(*	SINT_T, USINT_T, INT_T, UINT_T, DINT_T, UDINT_T, 
				LINT_T, ULINT_T, REALT_T, LREAL_T*)
CASE TypeOfValue OF
	//VAR_TYPES.SINT_T:
	IBaseLibrary.TypeClass.TYPE_SINT:
		GetValueStringFaktor := SINT_TO_STRING(VALUE.SINT_T);
	//VAR_TYPES.USINT_T:
	IBaseLibrary.TypeClass.TYPE_USINT:
		GetValueStringFaktor := USINT_TO_STRING(VALUE.USINT_T);		
	//VAR_TYPES.INT_T:
	IBaseLibrary.TypeClass.TYPE_INT:
		GetValueStringFaktor := INT_TO_STRING(VALUE.INT_T);
	//VAR_TYPES.UINT_T:
	IBaseLibrary.TypeClass.TYPE_UINT:
		GetValueStringFaktor := UINT_TO_STRING(VALUE.UINT_T);
	//VAR_TYPES.DINT_T:
	IBaseLibrary.TypeClass.TYPE_DINT:
		GetValueStringFaktor := DINT_TO_STRING(VALUE.DINT_T);
	//VAR_TYPES.UDINT_T:
	IBaseLibrary.TypeClass.TYPE_UDINT:
		GetValueStringFaktor := UDINT_TO_STRING(VALUE.UDINT_T);
	//VAR_TYPES.LINT_T:
	IBaseLibrary.TypeClass.TYPE_LINT:
		GetValueStringFaktor := LINT_TO_STRING(VALUE.LINT_T);
	//VAR_TYPES.ULINT_T:
	IBaseLibrary.TypeClass.TYPE_ULINT:
		GetValueStringFaktor := ULINT_TO_STRING(VALUE.ULINT_T);
	//VAR_TYPES.REAL_T:
	IBaseLibrary.TypeClass.TYPE_REAL:
		GetValueStringFaktor := OSCAT_BASIC.REAL_TO_STRF(VALUE.REAL_T * RealFaktor,DecimalPlace,'.');
	//VAR_TYPES.LREAL_T:
	IBaseLibrary.TypeClass.TYPE_LREAL:
		GetValueStringFaktor := BASIC_Extension.LREAL_TO_STRF(VALUE.LREAL_T * RealFaktor,DecimalPlace,'.');
	//VAR_TYPES.BYTE_T:
	IBaseLibrary.TypeClass.TYPE_BYTE:
		GetValueStringFaktor := BYTE_TO_STRING(VALUE.BYTE_T);
	//VAR_TYPES.WORD_T:
	IBaseLibrary.TypeClass.TYPE_WORD:
		GetValueStringFaktor := WORD_TO_STRING(VALUE.WORD_T);
	//VAR_TYPES.DWORD_T:
	IBaseLibrary.TypeClass.TYPE_DWORD:
		GetValueStringFaktor := DWORD_TO_STRING(VALUE.DWORD_T);
	//VAR_TYPES.LWORD_T:
	IBaseLibrary.TypeClass.TYPE_LWORD:
		GetValueStringFaktor := LWORD_TO_STRING(VALUE.LWORD_T);
	//VAR_TYPES.DT_T:
	IBaseLibrary.TypeClass.TYPE_DATEANDTIME:
		GetValueStringFaktor := DT_TO_STRING(VALUE.DT_T);
	//VAR_TYPES.TIME_T:
	IBaseLibrary.TypeClass.TYPE_TIME:
		GetValueStringFaktor := TIME_TO_STRING(VALUE.TIME_T);
	//VAR_TYPES.LTIME_T:
	IBaseLibrary.TypeClass.TYPE_LTIME:
		GetValueStringFaktor := LTIME_TO_STRING(VALUE.LTIME_T);
	//VAR_TYPES.TOD_T:
	IBaseLibrary.TypeClass.TYPE_TIMEOFDAY:
		GetValueStringFaktor := TOD_TO_STRING(VALUE.TOD_T);
	//VAR_TYPES.BOOL_T:
	IBaseLibrary.TypeClass.TYPE_BOOL:
		GetValueStringFaktor := BOOL_TO_STRING(VALUE.BOOL_T);
	//VAR_TYPES.DATE_T:
	IBaseLibrary.TypeClass.TYPE_DATE:
		GetValueStringFaktor := DATE_TO_STRING(VALUE.DATE_T);
END_CASE

END_FUNCTION

// Common/Functions/unionAdd
FUNCTION unionAdd : ALL_TYPES_UNION
VAR_INPUT
	a:ALL_TYPES_UNION;
	b:ALL_TYPES_UNION;
	TypeOfValue:IBaseLibrary.TypeClass;
END_VAR
VAR
END_VAR

(*	SINT_T, USINT_T, INT_T, UINT_T, DINT_T, UDINT_T, 
				LINT_T, ULINT_T, REALT_T, LREAL_T*)
CASE TypeOfValue OF
	IBaseLibrary.TypeClass.TYPE_SINT:
		unionAdd.SINT_T := a.SINT_T + b.SINT_T;
	IBaseLibrary.TypeClass.TYPE_USINT:
		unionAdd.USINT_T := a.USINT_T + b.USINT_T;
	IBaseLibrary.TypeClass.TYPE_INT:
		unionAdd.INT_T := a.INT_T + b.INT_T;
	IBaseLibrary.TypeClass.TYPE_UINT:
		unionAdd.UINT_T := a.UINT_T + b.UINT_T;
	IBaseLibrary.TypeClass.TYPE_DINT:
		unionAdd.DINT_T := a.UINT_T + b.UINT_T;
	IBaseLibrary.TypeClass.TYPE_UDINT:
		unionAdd.UDINT_T := a.UDINT_T + b.UDINT_T;
	IBaseLibrary.TypeClass.TYPE_LINT:
		unionAdd.LINT_T := a.LINT_T + b.LINT_T;
	IBaseLibrary.TypeClass.TYPE_ULINT:
		unionAdd.ULINT_T := a.ULINT_T + b.ULINT_T;
	IBaseLibrary.TypeClass.TYPE_REAL:
		unionAdd.REAL_T := a.REAL_T + b.REAL_T;
	IBaseLibrary.TypeClass.TYPE_LREAL:
		unionAdd.LREAL_T := a.LREAL_T + b.LREAL_T;
	IBaseLibrary.TypeClass.TYPE_BYTE:
		unionAdd.BYTE_T := a.BYTE_T + b.BYTE_T;
	IBaseLibrary.TypeClass.TYPE_WORD:
		unionAdd.WORD_T := a.WORD_T + b.WORD_T;
	IBaseLibrary.TypeClass.TYPE_DWORD:
		unionAdd.DWORD_T := a.DWORD_T + b.DWORD_T;
	IBaseLibrary.TypeClass.TYPE_LWORD:
		unionAdd.LWORD_T := a.LWORD_T + b.LWORD_T;
	IBaseLibrary.TypeClass.TYPE_DATEANDTIME:
	{warning "need to implement"}
		//unionAdd.DT_T := a.DT_T + b.DT_T;
	IBaseLibrary.TypeClass.TYPE_TIME:
		unionAdd.TIME_T := a.TIME_T + b.TIME_T;
	IBaseLibrary.TypeClass.TYPE_LTIME:
		unionAdd.LTIME_T := a.LTIME_T + b.LTIME_T;
	IBaseLibrary.TypeClass.TYPE_TIMEOFDAY:
	{warning "need to implement"}
		//unionAdd.TOD_T := a.TOD_T + b.TOD_T;
	IBaseLibrary.TypeClass.TYPE_BOOL:
		unionAdd.BOOL_T := a.BOOL_T AND b.BOOL_T;
	IBaseLibrary.TypeClass.TYPE_DATE:
	{warning "need to implement"}
		//unionAdd.DATE_T := a.DATE_T + b.DATE_T;
	
END_CASE

END_FUNCTION

// Common/Functions/unionSub
FUNCTION unionSub : ALL_TYPES_UNION
VAR_INPUT
	a:ALL_TYPES_UNION;
	b:ALL_TYPES_UNION;
	TypeOfValue:IBaseLibrary.TypeClass;
END_VAR
VAR
END_VAR

(*	SINT_T, USINT_T, INT_T, UINT_T, DINT_T, UDINT_T, 
				LINT_T, ULINT_T, REALT_T, LREAL_T*)
CASE TypeOfValue OF
	IBaseLibrary.TypeClass.TYPE_SINT:
		unionSub.SINT_T := a.SINT_T - b.SINT_T;
	IBaseLibrary.TypeClass.TYPE_USINT:
		unionSub.USINT_T := a.USINT_T - b.USINT_T;
	IBaseLibrary.TypeClass.TYPE_INT:
		unionSub.INT_T := a.INT_T - b.INT_T;
	IBaseLibrary.TypeClass.TYPE_UINT:
		unionSub.UINT_T := a.UINT_T - b.UINT_T;
	IBaseLibrary.TypeClass.TYPE_DINT:
		unionSub.DINT_T := a.UINT_T - b.UINT_T;
	IBaseLibrary.TypeClass.TYPE_UDINT:
		unionSub.UDINT_T := a.UDINT_T - b.UDINT_T;
	IBaseLibrary.TypeClass.TYPE_LINT:
		unionSub.LINT_T := a.LINT_T - b.LINT_T;
	IBaseLibrary.TypeClass.TYPE_ULINT:
		unionSub.ULINT_T := a.ULINT_T - b.ULINT_T;
	IBaseLibrary.TypeClass.TYPE_REAL:
		unionSub.REAL_T := a.REAL_T - b.REAL_T;
	IBaseLibrary.TypeClass.TYPE_LREAL:
		unionSub.LREAL_T := a.LREAL_T - b.LREAL_T;
	IBaseLibrary.TypeClass.TYPE_BYTE:
		unionSub.BYTE_T := a.BYTE_T - b.BYTE_T;
	IBaseLibrary.TypeClass.TYPE_WORD:
		unionSub.WORD_T := a.WORD_T - b.WORD_T;
	IBaseLibrary.TypeClass.TYPE_DWORD:
		unionSub.DWORD_T := a.DWORD_T - b.DWORD_T;
	IBaseLibrary.TypeClass.TYPE_LWORD:
		unionSub.LWORD_T := a.LWORD_T - b.LWORD_T;
	IBaseLibrary.TypeClass.TYPE_DATEANDTIME:
	{warning "need to implement"}
		//unionSub.DT_T := a.DT_T - b.DT_T;
	IBaseLibrary.TypeClass.TYPE_TIME:
		unionSub.TIME_T := a.TIME_T - b.TIME_T;
	IBaseLibrary.TypeClass.TYPE_LTIME:
		unionSub.LTIME_T := a.LTIME_T - b.LTIME_T;
	IBaseLibrary.TypeClass.TYPE_TIMEOFDAY:
	{warning "need to implement"}
		//unionSub.TOD_T := a.TOD_T - b.TOD_T;
	IBaseLibrary.TypeClass.TYPE_BOOL:
		unionSub.BOOL_T := a.BOOL_T AND b.BOOL_T;
	IBaseLibrary.TypeClass.TYPE_DATE:
	{warning "need to implement"}
		//unionSub.DATE_T := a.DATE_T - b.DATE_T;
	
END_CASE

END_FUNCTION

// Common/Functions/unionMul
FUNCTION unionMul : ALL_TYPES_UNION
VAR_INPUT
	a:ALL_TYPES_UNION;
	b:ALL_TYPES_UNION;
	TypeOfValue:IBaseLibrary.TypeClass;
END_VAR
VAR
END_VAR

(*	SINT_T, USINT_T, INT_T, UINT_T, DINT_T, UDINT_T, 
				LINT_T, ULINT_T, REALT_T, LREAL_T*)
CASE TypeOfValue OF
	IBaseLibrary.TypeClass.TYPE_SINT:
		unionMul.SINT_T := a.SINT_T * b.SINT_T;
	IBaseLibrary.TypeClass.TYPE_USINT:
		unionMul.USINT_T := a.USINT_T * b.USINT_T;
	IBaseLibrary.TypeClass.TYPE_INT:
		unionMul.INT_T := a.INT_T * b.INT_T;
	IBaseLibrary.TypeClass.TYPE_UINT:
		unionMul.UINT_T := a.UINT_T * b.UINT_T;
	IBaseLibrary.TypeClass.TYPE_DINT:
		unionMul.DINT_T := a.UINT_T * b.UINT_T;
	IBaseLibrary.TypeClass.TYPE_UDINT:
		unionMul.UDINT_T := a.UDINT_T * b.UDINT_T;
	IBaseLibrary.TypeClass.TYPE_LINT:
		unionMul.LINT_T := a.LINT_T * b.LINT_T;
	IBaseLibrary.TypeClass.TYPE_ULINT:
		unionMul.ULINT_T := a.ULINT_T * b.ULINT_T;
	IBaseLibrary.TypeClass.TYPE_REAL:
		unionMul.REAL_T := a.REAL_T * b.REAL_T;
	IBaseLibrary.TypeClass.TYPE_LREAL:
		unionMul.LREAL_T := a.LREAL_T * b.LREAL_T;
	IBaseLibrary.TypeClass.TYPE_BYTE:
		unionMul.BYTE_T := a.BYTE_T * b.BYTE_T;
	IBaseLibrary.TypeClass.TYPE_WORD:
		unionMul.WORD_T := a.WORD_T * b.WORD_T;
	IBaseLibrary.TypeClass.TYPE_DWORD:
		unionMul.DWORD_T := a.DWORD_T * b.DWORD_T;
	IBaseLibrary.TypeClass.TYPE_LWORD:
		unionMul.LWORD_T := a.LWORD_T * b.LWORD_T;
	IBaseLibrary.TypeClass.TYPE_DATEANDTIME:
	{warning "need to implement"}
		//unionMul.DT_T := a.DT_T * b.DT_T;
	IBaseLibrary.TypeClass.TYPE_TIME:
	//unionMul.TOD_T := a.TOD_T * b.TOD_T;
		//unionMul.TIME_T := a.TIME_T * b.TIME_T;
	IBaseLibrary.TypeClass.TYPE_LTIME:
	//unionMul.TOD_T := a.TOD_T * b.TOD_T;
		//unionMul.LTIME_T := a.LTIME_T * b.LTIME_T;
	IBaseLibrary.TypeClass.TYPE_TIMEOFDAY:
	{warning "need to implement"}
		//unionMul.TOD_T := a.TOD_T * b.TOD_T;
	IBaseLibrary.TypeClass.TYPE_BOOL:
		unionMul.BOOL_T := a.BOOL_T AND b.BOOL_T;
	IBaseLibrary.TypeClass.TYPE_DATE:
	{warning "need to implement"}
		//unionMul.DATE_T := a.DATE_T * b.DATE_T;
	
END_CASE

END_FUNCTION

// Common/Functions/unionDiv
FUNCTION unionDiv : ALL_TYPES_UNION
VAR_INPUT
	a:ALL_TYPES_UNION;
	b:ALL_TYPES_UNION;
	TypeOfValue:IBaseLibrary.TypeClass;
END_VAR
VAR
END_VAR

(*	SINT_T, USINT_T, INT_T, UINT_T, DINT_T, UDINT_T, 
				LINT_T, ULINT_T, REALT_T, LREAL_T*)
CASE TypeOfValue OF
	IBaseLibrary.TypeClass.TYPE_SINT:
		unionDiv.SINT_T := a.SINT_T / b.SINT_T;
	IBaseLibrary.TypeClass.TYPE_USINT:
		unionDiv.USINT_T := a.USINT_T / b.USINT_T;
	IBaseLibrary.TypeClass.TYPE_INT:
		unionDiv.INT_T := a.INT_T / b.INT_T;
	IBaseLibrary.TypeClass.TYPE_UINT:
		unionDiv.UINT_T := a.UINT_T / b.UINT_T;
	IBaseLibrary.TypeClass.TYPE_DINT:
		unionDiv.DINT_T := a.UINT_T / b.UINT_T;
	IBaseLibrary.TypeClass.TYPE_UDINT:
		unionDiv.UDINT_T := a.UDINT_T / b.UDINT_T;
	IBaseLibrary.TypeClass.TYPE_LINT:
		unionDiv.LINT_T := a.LINT_T / b.LINT_T;
	IBaseLibrary.TypeClass.TYPE_ULINT:
		unionDiv.ULINT_T := a.ULINT_T / b.ULINT_T;
	IBaseLibrary.TypeClass.TYPE_REAL:
		unionDiv.REAL_T := a.REAL_T / b.REAL_T;
	IBaseLibrary.TypeClass.TYPE_LREAL:
		unionDiv.LREAL_T := a.LREAL_T / b.LREAL_T;
	IBaseLibrary.TypeClass.TYPE_BYTE:
		unionDiv.BYTE_T := a.BYTE_T / b.BYTE_T;
	IBaseLibrary.TypeClass.TYPE_WORD:
		unionDiv.WORD_T := a.WORD_T / b.WORD_T;
	IBaseLibrary.TypeClass.TYPE_DWORD:
		unionDiv.DWORD_T := a.DWORD_T / b.DWORD_T;
	IBaseLibrary.TypeClass.TYPE_LWORD:
		unionDiv.LWORD_T := a.LWORD_T / b.LWORD_T;
	IBaseLibrary.TypeClass.TYPE_DATEANDTIME:
	{warning "need to implement"}
		//unionDiv.DT_T := a.DT_T / b.DT_T;
	IBaseLibrary.TypeClass.TYPE_TIME:
	//unionDiv.TOD_T := a.TOD_T / b.TOD_T;
		//unionDiv.TIME_T := a.TIME_T / b.TIME_T;
	IBaseLibrary.TypeClass.TYPE_LTIME:
	//unionDiv.TOD_T := a.TOD_T / b.TOD_T;
		//unionDiv.LTIME_T := a.LTIME_T / b.LTIME_T;
	IBaseLibrary.TypeClass.TYPE_TIMEOFDAY:
	{warning "need to implement"}
		//unionDiv.TOD_T := a.TOD_T / b.TOD_T;
	IBaseLibrary.TypeClass.TYPE_BOOL:
		unionDiv.BOOL_T := a.BOOL_T AND b.BOOL_T;
	IBaseLibrary.TypeClass.TYPE_DATE:
	{warning "need to implement"}
		//unionDiv.DATE_T := a.DATE_T / b.DATE_T;
	
END_CASE

END_FUNCTION

// Common/Function Blocks/UpDown
FUNCTION_BLOCK UpDown
VAR_INPUT
	Start:BOOL;
	VarType:IBaseLibrary.TypeClass;
	faktor:UINT;
	Imp: BOOL;
	limitUp:REAL;
	limitDown:REAL;
END_VAR
VAR_IN_OUT
	Who:ALL_TYPES_UNION;
	
END_VAR
VAR_OUTPUT
END_VAR
VAR
	dir: BOOL;
	triggerStart:R_TRIG;
	diffVal:ALL_TYPES_UNION;
END_VAR

triggerStart(CLK := Start);
IF triggerStart.Q THEN
	dir := NOT dir;
END_IF

IF Start AND Imp THEN
	diffVal := uint_to_Union(value:= faktor, TypeOfValue:= VarType);
	IF dir THEN
		who := unionAdd(a:= Who, b:= diffVal, TypeOfValue:= VarType);
	ELSE
		who := unionSub(a:= Who, b:= diffVal, TypeOfValue:= VarType);
	END_IF
END_IF

END_FUNCTION_BLOCK

// Common/Functions/uint_to_Union
FUNCTION uint_to_Union : ALL_TYPES_UNION
VAR_INPUT
	TypeOfValue:IBaseLibrary.TypeClass;
	value:UINT;	

END_VAR
VAR
END_VAR

(*	SINT_T, USINT_T, INT_T, UINT_T, DINT_T, UDINT_T, 
				LINT_T, ULINT_T, REALT_T, LREAL_T*)
CASE TypeOfValue OF
	IBaseLibrary.TypeClass.TYPE_SINT:
		uint_to_Union.SINT_T := TO_SINT(value);
	IBaseLibrary.TypeClass.TYPE_USINT:
		uint_to_Union.USINT_T := TO_USINT(value);		
	IBaseLibrary.TypeClass.TYPE_INT:
		uint_to_Union.INT_T := TO_INT(value);
	IBaseLibrary.TypeClass.TYPE_UINT:
		uint_to_Union.UINT_T := TO_UINT(value);
	IBaseLibrary.TypeClass.TYPE_DINT:
		uint_to_Union.DINT_T := TO_DINT(value);
	IBaseLibrary.TypeClass.TYPE_UDINT:
		uint_to_Union.UDINT_T := TO_UDINT(value);
	IBaseLibrary.TypeClass.TYPE_LINT:
		AtomicWriteLInt(pDest:= ADR(uint_to_Union.LINT_T), liValue:= TO_LINT(value));
	IBaseLibrary.TypeClass.TYPE_ULINT:
		AtomicWriteULInt(pDest:= ADR(uint_to_Union.ULINT_T), uliValue:= TO_ULINT(value));
	IBaseLibrary.TypeClass.TYPE_REAL:
		uint_to_Union.REAL_T := TO_REAL(value);
	IBaseLibrary.TypeClass.TYPE_LREAL:
		AtomicWriteLReal(pDest:= ADR(uint_to_Union.LREAL_T), lrValue:= TO_LREAL(value));
	IBaseLibrary.TypeClass.TYPE_BYTE:
		uint_to_Union.BYTE_T := TO_BYTE(value);
	IBaseLibrary.TypeClass.TYPE_WORD:
		uint_to_Union.WORD_T := TO_WORD(value);
	IBaseLibrary.TypeClass.TYPE_DWORD:
		uint_to_Union.DWORD_T := TO_DWORD(value);
	IBaseLibrary.TypeClass.TYPE_LWORD:
		AtomicWriteLWord(pDest:= ADR(uint_to_Union.LWORD_T), lwValue:= TO_LWORD(value));
	IBaseLibrary.TypeClass.TYPE_DATEANDTIME:
		uint_to_Union.DT_T := TO_DT(value);
	IBaseLibrary.TypeClass.TYPE_TIME:
		uint_to_Union.TIME_T := TO_TIME(value);
	IBaseLibrary.TypeClass.TYPE_LTIME:
		AtomicWriteLTime(pDest:= ADR(uint_to_Union.LTIME_T), ltValue:= TO_LTIME(value));
	IBaseLibrary.TypeClass.TYPE_TIMEOFDAY:
		uint_to_Union.TOD_T := TO_TOD(value);
	IBaseLibrary.TypeClass.TYPE_BOOL:
		uint_to_Union.BOOL_T := TO_BOOL(value);
	IBaseLibrary.TypeClass.TYPE_DATE:
		uint_to_Union.DATE_T := TO_DATE(value);
	
	
END_CASE

END_FUNCTION

// Common/Functions/unionLimit
FUNCTION unionLimit : ALL_TYPES_UNION
VAR_INPUT
	in:ALL_TYPES_UNION;
	lMin:ALL_TYPES_UNION;
	lMax:ALL_TYPES_UNION;
	TypeOfValue:IBaseLibrary.TypeClass;
END_VAR
VAR
END_VAR

(*	SINT_T, USINT_T, INT_T, UINT_T, DINT_T, UDINT_T, 
				LINT_T, ULINT_T, REALT_T, LREAL_T*)
CASE TypeOfValue OF
	IBaseLibrary.TypeClass.TYPE_SINT:
		unionLimit.SINT_T := LIMIT(lMin.SINT_T, IN.SINT_T, lMax.SINT_T);
	IBaseLibrary.TypeClass.TYPE_USINT:
		unionLimit.USINT_T := LIMIT(lMin.USINT_T, IN.USINT_T, lMax.USINT_T);
	IBaseLibrary.TypeClass.TYPE_INT:
		unionLimit.INT_T := LIMIT(lMin.INT_T, IN.INT_T, lMax.INT_T);
	IBaseLibrary.TypeClass.TYPE_UINT:
		unionLimit.UINT_T := LIMIT(lMin.UINT_T, IN.UINT_T, lMax.UINT_T);
	IBaseLibrary.TypeClass.TYPE_DINT:
		unionLimit.DINT_T := LIMIT(lMin.DINT_T, IN.DINT_T, lMax.DINT_T);
	IBaseLibrary.TypeClass.TYPE_UDINT:
		unionLimit.UDINT_T := LIMIT(lMin.UDINT_T, IN.UDINT_T, lMax.UDINT_T);
	IBaseLibrary.TypeClass.TYPE_LINT:
		unionLimit.LINT_T := LIMIT(lMin.LINT_T, IN.LINT_T, lMax.LINT_T);
	IBaseLibrary.TypeClass.TYPE_ULINT:
		unionLimit.ULINT_T := LIMIT(lMin.ULINT_T, IN.ULINT_T, lMax.ULINT_T);
	IBaseLibrary.TypeClass.TYPE_REAL:
		unionLimit.REAL_T := LIMIT(lMin.REAL_T, IN.REAL_T, lMax.REAL_T);
	IBaseLibrary.TypeClass.TYPE_LREAL:
		unionLimit.LREAL_T := LIMIT(lMin.LREAL_T, IN.LREAL_T, lMax.LREAL_T);
	IBaseLibrary.TypeClass.TYPE_BYTE:
		unionLimit.BYTE_T := LIMIT(lMin.BYTE_T, IN.BYTE_T, lMax.BYTE_T);
	IBaseLibrary.TypeClass.TYPE_WORD:
		unionLimit.WORD_T := LIMIT(lMin.WORD_T, IN.WORD_T, lMax.WORD_T);
	IBaseLibrary.TypeClass.TYPE_DWORD:
		unionLimit.DWORD_T := LIMIT(lMin.DWORD_T, IN.DWORD_T, lMax.DWORD_T);
	IBaseLibrary.TypeClass.TYPE_LWORD:
		unionLimit.LWORD_T := LIMIT(lMin.LWORD_T, IN.LWORD_T, lMax.LWORD_T);
	IBaseLibrary.TypeClass.TYPE_DATEANDTIME:
		unionLimit.DT_T := LIMIT(lMin.DT_T, IN.DT_T, lMax.DT_T);
	IBaseLibrary.TypeClass.TYPE_TIME:
		unionLimit.TIME_T := LIMIT(lMin.TIME_T, IN.TIME_T, lMax.TIME_T);
	IBaseLibrary.TypeClass.TYPE_LTIME:
		unionLimit.LTIME_T := LIMIT(lMin.LTIME_T, IN.LTIME_T, lMax.LTIME_T);
	IBaseLibrary.TypeClass.TYPE_TIMEOFDAY:
		unionLimit.TOD_T := LIMIT(lMin.TOD_T, IN.TOD_T, lMax.TOD_T);
	IBaseLibrary.TypeClass.TYPE_BOOL:
		unionLimit.BOOL_T := LIMIT(lMin.BOOL_T, IN.BOOL_T, lMax.BOOL_T);
	IBaseLibrary.TypeClass.TYPE_DATE:
		unionLimit.DATE_T := LIMIT(lMin.DATE_T, IN.DATE_T, lMax.DATE_T);
	
END_CASE

END_FUNCTION

// Common/Functions/ScaleAllTypesUnion
FUNCTION ScaleAllTypesUnion : ALL_TYPES_UNION
VAR_INPUT
	in:ALL_TYPES_UNION;
	TypeOfVar:IBaseLibrary.TypeClass;
	I_LO : LREAL;
	I_HI : LREAL;
	O_LO : LREAL;
	O_HI : LREAL;
END_VAR
VAR

END_VAR

(*	SINT_T, USINT_T, INT_T, UINT_T, DINT_T, UDINT_T, 
				LINT_T, ULINT_T, REALT_T, LREAL_T*)
CASE TypeOfVar OF
	IBaseLibrary.TypeClass.TYPE_SINT:
		ScaleAllTypesUnion.SINT_T := TO_SINT(OSCAT_BASIC.SCALE_D(
			X:= TO_DWORD(in.SINT_T), I_LO:= TO_DWORD(I_LO), I_HI:= TO_DWORD(I_HI), O_LO:= TO_REAL(O_LO), O_HI:= TO_REAL(O_HI)));
	IBaseLibrary.TypeClass.TYPE_USINT:
		ScaleAllTypesUnion.USINT_T := TO_USINT(OSCAT_BASIC.SCALE_D(
			X:= TO_DWORD(in.USINT_T), I_LO:= TO_DWORD(I_LO), I_HI:= TO_DWORD(I_HI), O_LO:= TO_REAL(O_LO), O_HI:= TO_REAL(O_HI)));
	IBaseLibrary.TypeClass.TYPE_INT:
		ScaleAllTypesUnion.INT_T := TO_INT(OSCAT_BASIC.SCALE_D(
			X:= TO_DWORD(in.INT_T), I_LO:= TO_DWORD(I_LO), I_HI:= TO_DWORD(I_HI), O_LO:= TO_REAL(O_LO), O_HI:= TO_REAL(O_HI)));
	IBaseLibrary.TypeClass.TYPE_UINT:
		ScaleAllTypesUnion.UINT_T := TO_UINT(OSCAT_BASIC.SCALE_D(
			X:= TO_DWORD(in.UINT_T), I_LO:= TO_DWORD(I_LO), I_HI:= TO_DWORD(I_HI), O_LO:= TO_REAL(O_LO), O_HI:= TO_REAL(O_HI)));
	IBaseLibrary.TypeClass.TYPE_DINT:
		ScaleAllTypesUnion.DINT_T := TO_DINT(OSCAT_BASIC.SCALE_D(
			X:= TO_DWORD(in.DINT_T), I_LO:= TO_DWORD(I_LO), I_HI:= TO_DWORD(I_HI), O_LO:= TO_REAL(O_LO), O_HI:= TO_REAL(O_HI)));
	IBaseLibrary.TypeClass.TYPE_UDINT:
		ScaleAllTypesUnion.UDINT_T := TO_UDINT(OSCAT_BASIC.SCALE_D(
			X:= TO_DWORD(in.UDINT_T), I_LO:= TO_DWORD(I_LO), I_HI:= TO_DWORD(I_HI), O_LO:= TO_REAL(O_LO), O_HI:= TO_REAL(O_HI)));
	IBaseLibrary.TypeClass.TYPE_LINT:
		ScaleAllTypesUnion.LINT_T := TO_LINT(BASIC_Extension.SCALE_L(
			X:= TO_DWORD(in.LINT_T), I_LO:= TO_DWORD(I_LO), I_HI:= TO_DWORD(I_HI), O_LO:= TO_REAL(O_LO), O_HI:= TO_REAL(O_HI)));
	IBaseLibrary.TypeClass.TYPE_ULINT:
		ScaleAllTypesUnion.ULINT_T := TO_ULINT(BASIC_Extension.SCALE_L(
			X:= TO_DWORD(in.ULINT_T), I_LO:= TO_DWORD(I_LO), I_HI:= TO_DWORD(I_HI), O_LO:= TO_REAL(O_LO), O_HI:= TO_REAL(O_HI)));
	IBaseLibrary.TypeClass.TYPE_REAL:
		ScaleAllTypesUnion.REAL_T := OSCAT_BASIC.SCALE_R(
			X:= in.REAL_T, I_LO:= TO_REAL(I_LO), I_HI:= TO_REAL(I_HI), O_LO:= TO_REAL(O_LO), O_HI:= TO_REAL(O_HI));
	IBaseLibrary.TypeClass.TYPE_LREAL:
		ScaleAllTypesUnion.LREAL_T := BASIC_Extension.SCALE_LR(
			X:= in.LREAL_T, I_LO:= I_LO, I_HI:= I_HI, O_LO:= O_LO, O_HI:= O_HI);
	IBaseLibrary.TypeClass.TYPE_BYTE:
		ScaleAllTypesUnion.BYTE_T := TO_BYTE(OSCAT_BASIC.SCALE_B(
			X:= in.BYTE_T, I_LO:= TO_BYTE(I_LO), I_HI:= TO_BYTE(I_HI), O_LO:= TO_REAL(O_LO), O_HI:= TO_REAL(O_HI)));
	IBaseLibrary.TypeClass.TYPE_WORD:
		ScaleAllTypesUnion.WORD_T := TO_WORD(OSCAT_BASIC.SCALE_D(
			X:= TO_DWORD(in.WORD_T), I_LO:= TO_DWORD(I_LO), I_HI:= TO_DWORD(I_HI), O_LO:= TO_REAL(O_LO), O_HI:= TO_REAL(O_HI)));
	IBaseLibrary.TypeClass.TYPE_DWORD:
		ScaleAllTypesUnion.DWORD_T := TO_DWORD(OSCAT_BASIC.SCALE_D(
			X:= in.DWORD_T, I_LO:= TO_DWORD(I_LO), I_HI:= TO_DWORD(I_HI), O_LO:= TO_REAL(O_LO), O_HI:= TO_REAL(O_HI)));
	IBaseLibrary.TypeClass.TYPE_LWORD:
		ScaleAllTypesUnion.LWORD_T := TO_LWORD(BASIC_Extension.SCALE_L(
			X:= in.LWORD_T, I_LO:= TO_LWORD(I_LO), I_HI:= TO_LWORD(I_HI), O_LO:= O_LO, O_HI:= O_HI));
	IBaseLibrary.TypeClass.TYPE_DATEANDTIME:
		ScaleAllTypesUnion.DT_T := TO_DT(OSCAT_BASIC.SCALE_D(
			X:= TO_DWORD(in.DT_T), I_LO:= TO_DWORD(I_LO), I_HI:= TO_DWORD(I_HI), O_LO:= TO_REAL(O_LO), O_HI:= TO_REAL(O_HI)));
	IBaseLibrary.TypeClass.TYPE_TIME:
		ScaleAllTypesUnion.TIME_T := TO_TIME(OSCAT_BASIC.SCALE_D(
			X:= TO_DWORD(in.TIME_T), I_LO:= TO_DWORD(I_LO), I_HI:= TO_DWORD(I_HI), O_LO:= TO_REAL(O_LO), O_HI:= TO_REAL(O_HI)));
	IBaseLibrary.TypeClass.TYPE_LTIME:
		ScaleAllTypesUnion.LTIME_T := TO_LTIME(BASIC_Extension.SCALE_L(
			X:= TO_LWORD(in.LTIME_T), I_LO:= TO_LWORD(I_LO), I_HI:= TO_LWORD(I_HI), O_LO:= O_LO, O_HI:= O_HI));
	IBaseLibrary.TypeClass.TYPE_TIMEOFDAY:
		ScaleAllTypesUnion.TOD_T := TO_TOD(OSCAT_BASIC.SCALE_D(
			X:= TO_DWORD(in.TOD_T), I_LO:= TO_DWORD(I_LO), I_HI:= TO_DWORD(I_HI), O_LO:= TO_REAL(O_LO), O_HI:= TO_REAL(O_HI)));
	IBaseLibrary.TypeClass.TYPE_BOOL:
		ScaleAllTypesUnion.BOOL_T := in.BOOL_T;
	IBaseLibrary.TypeClass.TYPE_DATE:
		ScaleAllTypesUnion.DATE_T := TO_DATE(OSCAT_BASIC.SCALE_D(
			X:= TO_DWORD(in.DATE_T), I_LO:= TO_DWORD(I_LO), I_HI:= TO_DWORD(I_HI), O_LO:= TO_REAL(O_LO), O_HI:= TO_REAL(O_HI)));
END_CASE

END_FUNCTION

// Common/Function Blocks/BLIND_INPUT_PERS
FUNCTION_BLOCK BLIND_INPUT_PERS
VAR_INPUT
	POS, ANG : BYTE;
	S1, S2 : BOOL;
	IN : BOOL;
	PI, AI : BYTE;
END_VAR
VAR_INPUT CONSTANT
	SINGLE_SWITCH : BOOL;
	CLICK_EN : BOOL := TRUE;
	CLICK_TIME : TIME := T#500ms;
	MAX_RUNTIME : TIME := T#60s;
	MANUAL_TIMEOUT: TIME := T#1h;
	DEBOUNCE_TIME : TIME := T#20ms;
	DBL_CLK1 : BOOL := FALSE;
	DBL_POS1 : BYTE;
	DBL_ANG1 : BYTE;
	DBL_CLK2 : BOOL := FALSE;
	DBL_POS2 : BYTE := 255;
	DBL_ANG2 : BYTE := 255;
	D1_TOGGLE : BOOL := TRUE;
	D2_TOGGLE : BOOL := TRUE;
	MASTER_MODE : BOOL;
END_VAR
VAR_OUTPUT
	QU : BOOL := TRUE;
	QD : BOOL := TRUE;
	STATUS : BYTE;
	PO : BYTE := 255;
	AO : BYTE := 255;
	D1, D2 : BOOL;
END_VAR
VAR
	s1e, s2e : OSCAT_BASIC.TOF;
	s1d, s2d : OSCAT_BUILDING.CLICK_MODE;
	dir : BOOL;
	tx, last : TIME;
END_VAR
VAR PERSISTENT RETAIN
	_STATUS:BYTE;
END_VAR

(*
version 1.7	12. nov. 2009
programmer 	hugo
tested by		oscat


*)

(* read system timer *)
tx := DWORD_TO_TIME(OSCAT_BASIC.T_PLC_MS());

(* inputs S1 and S2 are debounced and then decoded for multiple clicks *)
s1e(in := S1, pt := DEBOUNCE_TIME);
s2e(in := S2, pt := DEBOUNCE_TIME);
s1d(in := (s1e.Q AND NOT SINGLE_SWITCH) OR (s1e.Q AND SINGLE_SWITCH AND dir), t_long := CLICK_TIME);
s2d(in := (s2e.Q AND NOT SINGLE_SWITCH) OR (s1e.Q AND SINGLE_SWITCH AND NOT dir), t_long := CLICK_TIME);

(* if d1 and d2 are not toggle clear them to make sure they are only active for oine cycle *)
IF NOT d1_toggle THEN d1 := FALSE; END_IF;
IF NOT d2_toggle THEN d2 := FALSE; END_IF;

(* decode actions *)
IF (s1d.LONG AND s2d.LONG) OR (_status = 139) THEN
   _status := 139;
   IF NOT (s1d.LONG OR s2d.LONG)  THEN _status := 130; END_IF;
ELSIF s1d.tp_LONG THEN
	_status := 132;
ELSIF s2d.tp_LONG THEN
	_status := 133;
ELSIF  s1d.SINGLE THEN
	IF click_en THEN
		(* if running then we stop otherwise start new direction *)
		IF QU XOR QD THEN
			_status := 131;
		ELSE
			_status := 134;
			last := tx;
			dir := NOT dir;
		END_IF;
	END_IF;
ELSIF  s2d.SINGLE THEN
	IF click_en THEN
		(* if running then we stop otherwise start new direction *)
		IF QU XOR QD THEN
			_status := 131;
		ELSE
			_status := 135;
			last := tx;
			dir := NOT dir;
		END_IF;
	END_IF;
ELSIF in THEN
	_status := 136;
	last := tx;
ELSIF s1d.DOUBLE THEN
	IF dbl_clk1 THEN
		(* a position need to be set for a double click on S1 *)
		_status := 137;
		last := tx;
	ELSE
		(* toggle the output when dbl_clk1 is not active *)
		D1 := NOT D1;
	END_IF;
ELSIF s2d.DOUBLE THEN
	IF dbl_clk2 THEN
		(* a position need to be set for a double click on S2 *)
		_status := 138;
		last := tx;
	ELSE
		(* toggle the output when dbl_clk2 is not active *)
		(* in single switch mode we need to toggle d1 instead of d2 *)
		IF single_switch THEN D1 := NOT D1; ELSE D2 := NOT D2; END_IF;
	END_IF;
END_IF;


(* state machine *)
CASE _status OF
	0:		(* power up operation *)
			_status := 130;

	130:	(* automatic operation standby *)
			IF NOT master_mode THEN
				PO := POS;
				AO := ANG;
			END_IF;
			QU := TRUE;
			QD := TRUE;

	131:	(* manual operation standby *)
			QU := FALSE;
			QD := FALSE;
			PO := POS;
			AO := ANG;
			(* manual mode will be ended when timeout is reached *)
			IF tx - last >= manual_timeout THEN
				_status := 130;
			END_IF;

	132:	(* manual operation up *)
			QU := TRUE;
			QD := FALSE;
			PO := POS; AO := ANG;
			last := tx;
			IF NOT s1d.LONG THEN _status := 131; dir := NOT dir; END_IF;

	133:	(* manual operation down *)
			QU := FALSE;
			QD := TRUE;
			PO := POS; AO := ANG;
			last := tx;
			IF NOT s2d.LONG THEN	_status := 131; dir := NOT dir; END_IF;

	134:	(* manual operation single click up *)
			QU := TRUE;
			QD := FALSE;
			PO := POS; AO := ANG;
			IF tx - last >= max_runtime THEN _status := 131; END_IF;

	135:	(* manual operation single click dn *)
			QU := FALSE;
			QD := TRUE;
			PO := POS; AO := ANG;
			IF tx - last >= max_runtime THEN _status := 131;	END_IF;

	136:	(* forced input in = true *)
			QU := TRUE;
			QD := TRUE;
			PO := PI; AO := AI;
			IF tx-last >= max_runtime THEN _status := 130; END_IF;

	137:	(* double click1 position *)
			QU := TRUE;
			QD := TRUE;
			PO := DBL_POS1;
			AO := DBL_ANG1;
			IF tx - last >= max_runtime THEN _status := 131; END_IF;

	138:	(* double click2 position *)
			QU := TRUE;
			QD := TRUE;
			PO := DBL_POS2;
			AO := DBL_ANG2;
			IF tx - last >= max_runtime THEN _status := 131; END_IF;

	   139:   (* manual operation standby *)
	         QU := FALSE;
	         QD := FALSE;
	         PO := POS;
	         AO := ANG;

END_CASE;

STATUS := _STATUS;

(* revision history
hm	29. sep 2007	rev 1.0
	original release

hm	6. oct 2007		rev 1.1
	renamed ps and as to po and ao

hm	30. dec 2007	rev 1.2
	added click_timeout variable and function

hm	16. jul. 2008	rev 1.3
	rewirtten code to allow for more functionality
	added single click mode with single_switch.
	added Debounce for inputs S1 and S2
	added double_click functionality

hm	26. sep. 2008	rev 1.4
	corrected an error while POS and ANG was transferred to outputs PO and AO during automatic modes

hm	22. jan 2009	rev 1.5
	added pulse mode for double click outputs
	added automatic mode for IN

hm	27. jul 2009	rev 1.6
	changed _status 0 to 130

HF	12. nov. 2009	rev 1.7
	added state 139
	set defaults for QU, QD, PO

*)

END_FUNCTION_BLOCK

// Common/Function Blocks/BLIND_CONTROL_S_PERS
FUNCTION_BLOCK BLIND_CONTROL_S_PERS
VAR_INPUT
	UP, DN : BOOL;
	S_IN : BYTE := 125;
	PI : BYTE;
	T_UP : TIME;
	T_DN : TIME;
	RU : BOOL;
	RD : BOOL;
END_VAR
VAR_INPUT CONSTANT
	T_LOCKOUT: TIME := T#100ms;
	T_EXT : TIME;
	EXT_TRIG : BYTE := 5;
	R_POS_TOP : BYTE := 255;
	R_POS_BOT : BYTE;
END_VAR
VAR_OUTPUT
	POS : BYTE;
	MU, MD : BOOL;
	STATUS : BYTE;
END_VAR
VAR
	rmp : OSCAT_BASIC._RMP_NEXT;
	tx, last : TIME;
	PI_last: BYTE;
END_VAR
VAR PERSISTENT RETAIN
	_STATUS:BYTE;
	_POS:BYTE;
END_VAR

(*
version 1.2	23. jan 2010
programmer 	hugo
tested by		heinz


*)


(* status definition
	121 = manual up				manual up operation UP = true and DN = false
	122 = manual down			manual down operation DN = true and UP = false
	123 = auto positioning		automatic mode DN = UP = TRUE
	124 = revert					revert from top or bottom
	125 = nothing					default input for S_IN
	127 = Lockout time			lockout between directional change
	128 = calibrate				calibrate after power up
	129 = extend					extend runtime at top or bottom for continuous calibration
*)

(* read system time *)
tx := DWORD_TO_TIME(OSCAT_BASIC.T_PLC_MS());

(* check inputs and start state machine *)
IF UP  AND NOT DN THEN
	(*  manual UP *)
	rmp.IN := 255;
	_STATUS := 121;
ELSIF DN AND NOT UP THEN
	(* manual DN *)
	rmp.IN := 0;
	_STATUS := 122;
ELSIF NOT (UP OR DN) THEN
	(* manual standby mode *)
	rmp.IN := PI;
	_STATUS := S_IN;
END_IF;

(* simulate pos output *)
rmp(E := UP OR DN, TR := T_UP, TF := T_DN, TL := T_LOCKOUT, OUT := _POS);

(* state machine *)
CASE _STATUS OF
	0:		(* power up init *)
		last := tx;
		PI_last := PI XOR BYTE#255;
		_STATUS := 128;		(* calibrate *)

	121: 	(* manual up *)
		MU := TRUE;
		MD := FALSE;
		IF _POS >= (BYTE#255 - EXT_TRIG) THEN
			(* extend cycle if top is reached *)
			_POS := 255;
			last := tx;
			_STATUS := 129;	(* extend *)
		END_IF;

	122:	(* manual down *)
		MD := TRUE;
		MU := FALSE;
		IF _POS <= EXT_TRIG THEN
			(* extend cycle if bottom is reached *)
			_POS := 0;
			last := tx;
			_STATUS := 129;	(* extend *)
		END_IF;

	123:	(* auto positioning *)
		MD := rmp.DN;
		MU := rmp.UP;
		IF NOT (rmp.DN OR rmp.UP) THEN
			(* automatic position is reached *)
			IF _POS <= EXT_TRIG THEN
				(* extend at bottom *)
				MD := TRUE;
				last := tx;
				_STATUS := 129;	(* extend *)
			ELSIF _POS >= (BYTE#255 - EXT_TRIG)  THEN
				(* extend at top *)
				MU := TRUE;
				last := tx;
				_STATUS := 129;	(* extend *)
			ELSE
				_STATUS := S_IN;
			END_IF;
		END_IF;

	124:	(* revert from top or bottom *)
		MD := rmp.DN;
		MU := rmp.UP;
		IF NOT(rmp.DN OR rmp.UP) THEN
(*		IF _POS = rmp.IN THEN  *)
			PI_last := PI;
			_STATUS := S_IN;
		END_IF;

	127:	(* lockout time *)
		IF (tx - last) >= T_LOCKOUT THEN
				_STATUS := S_IN;
		END_IF;

	128:	(* calibration *)
		MU := TRUE;
		MD := FALSE;
		rmp.IN := 255;
		IF (tx - last) >= (T_UP +  T_EXT) THEN
			MU := FALSE;
			last := tx;
			_STATUS := 127;	(* lockout *)
		END_IF;

	129: (* extend mode *)
		IF (tx - last) >= T_EXT THEN
			MU := FALSE;
			MD := FALSE;
			last := tx;
			_STATUS := 127;	(* lockout *)
		END_IF;

ELSE
	MU := FALSE;
	MD := FALSE;
	IF PI <> PI_last THEN
		PI_last := PI;
		rmp.IN := PI;
		_STATUS := 123;	(* auto positioning *)
	ELSIF _POS = 0 AND RU THEN
		rmp.IN := R_POS_BOT;
		_STATUS := 124;	(* revert *)
	ELSIF _POS = 255 AND RD THEN
		rmp.IN := R_POS_TOP;
		_STATUS := 124;	(* revert *)
	ELSE
		_STATUS := S_IN;
	END_IF;
END_CASE;

STATUS := _STATUS;
POS := _POS;
(* revision history

hm	9. mar. 2009	rev 1.0
	original release

hf	27. jul 2009	rev 1.1
	major code changes and updates

hf	23. Jan 2010	rev 1.2
	fixed a bug during calibration
	added T_UP and T_DN

*)

END_FUNCTION_BLOCK

// Common/Function Blocks/BLIND_INPUT_EXT_PERS
FUNCTION_BLOCK BLIND_INPUT_EXT_PERS
VAR_INPUT
	UP, DN: BOOL;
	POS, ANG : BYTE;
	S1, S2 : BOOL;
	IN : BOOL;
	PI, AI : BYTE;
	//S_IN:BYTE := 250;

END_VAR
VAR_INPUT CONSTANT
	SINGLE_SWITCH : BOOL;
	CLICK_EN : BOOL := TRUE;
	CLICK_TIME : TIME := T#500ms;
	MAX_RUNTIME : TIME := T#60s;
	MANUAL_TIMEOUT: TIME := T#1h;
	DEBOUNCE_TIME : TIME := T#20ms;
	DBL_CLK1 : BOOL := FALSE;
	DBL_POS1 : BYTE;
	DBL_ANG1 : BYTE;
	DBL_CLK2 : BOOL := FALSE;
	DBL_POS2 : BYTE := 255;
	DBL_ANG2 : BYTE := 255;
	D1_TOGGLE : BOOL := TRUE;
	D2_TOGGLE : BOOL := TRUE;
	MASTER_MODE : BOOL;
	NO_AUTO_AUTO: BOOL := FALSE;
END_VAR
VAR_OUTPUT
	QU : BOOL := TRUE;
	QD : BOOL := TRUE;
	STATUS : BYTE;
	PO : BYTE := 255;
	AO : BYTE := 255;
	D1, D2 : BOOL;
END_VAR
VAR
	s1e, s2e : OSCAT_BASIC.TOF;
	s1d, s2d : OSCAT_BUILDING.CLICK_MODE;
	dir : BOOL;
	tx, last : TIME;
	R1, R2:Standard.R_TRIG;
	startupDone: BOOL;

END_VAR
VAR PERSISTENT RETAIN
	_STATUS:BYTE;
END_VAR
(*
version 1.7	12. nov. 2009
programmer 	hugo
tested by		oscat


*)

(* read system timer *)
tx := DWORD_TO_TIME(OSCAT_BASIC.T_PLC_MS());

(* inputs S1 and S2 are debounced and then decoded for multiple clicks *)
s1e(in := S1, pt := DEBOUNCE_TIME);
s2e(in := S2, pt := DEBOUNCE_TIME);
s1d(in := (s1e.Q AND NOT SINGLE_SWITCH) OR (s1e.Q AND SINGLE_SWITCH AND dir), t_long := CLICK_TIME);
s2d(in := (s2e.Q AND NOT SINGLE_SWITCH) OR (s1e.Q AND SINGLE_SWITCH AND NOT dir), t_long := CLICK_TIME);

(* if d1 and d2 are not toggle clear them to make sure they are only active for oine cycle *)
IF NOT d1_toggle THEN d1 := FALSE; END_IF;
IF NOT d2_toggle THEN d2 := FALSE; END_IF;

(* decode actions *)
IF (s1d.LONG AND s2d.LONG) OR (_STATUS = 139) THEN
   _STATUS := 139;
   IF NOT (s1d.LONG OR s2d.LONG)  THEN _STATUS := 130; END_IF;
ELSIF s1d.tp_LONG THEN
	_STATUS := 132;
ELSIF s2d.tp_LONG THEN
	_STATUS := 133;
ELSIF  s1d.SINGLE THEN
	IF click_en THEN
		(* if running then we stop otherwise start new direction *)
		IF QU XOR QD THEN
			_STATUS := 131;
		ELSE
			_STATUS := 134;
			last := tx;
			dir := NOT dir;
		END_IF;
	END_IF;
ELSIF  s2d.SINGLE THEN
	IF click_en THEN
		(* if running then we stop otherwise start new direction *)
		IF QU XOR QD THEN
			_STATUS := 131;
		ELSE
			_STATUS := 135;
			last := tx;
			dir := NOT dir;
		END_IF;
	END_IF;
ELSIF in THEN
	_STATUS := 136;
	last := tx;
ELSIF s1d.DOUBLE THEN
	IF dbl_clk1 THEN
		(* a position need to be set for a double click on S1 *)
		_STATUS := 137;
		last := tx;
	ELSE
		(* toggle the output when dbl_clk1 is not active *)
		D1 := NOT D1;
	END_IF;
ELSIF s2d.DOUBLE THEN
	IF dbl_clk2 THEN
		(* a position need to be set for a double click on S2 *)
		_STATUS := 138;
		last := tx;
	ELSE
		(* toggle the output when dbl_clk2 is not active *)
		(* in single switch mode we need to toggle d1 instead of d2 *)
		IF single_switch THEN D1 := NOT D1; ELSE D2 := NOT D2; END_IF;
	END_IF;
END_IF;
R1(CLK:= DN);
R2(CLK:= UP);
IF R1.Q OR R2.Q THEN
	_STATUS := 130;
	startupDone := TRUE;
END_IF 

(* state machine *)
CASE _STATUS OF
	0:		(* power up operation *)
			IF NO_AUTO_AUTO THEN
				_STATUS := 131;
			ELSE
				_STATUS := 130;
			END_IF
			

	130:	(* automatic operation standby *)
			IF NOT master_mode THEN
				PO := POS;
				AO := ANG;
			END_IF;  
			IF NOT NO_AUTO_AUTO OR NOT startupDone THEN
				QU := TRUE;
				QD := TRUE;
			ELSE
				QU := UP;
				QD := DN;
			END_IF

	131:	(* manual operation standby *)
			QU := FALSE;
			QD := FALSE;
			PO := POS;
			AO := ANG;
			(* manual mode will be ended when timeout is reached *)
			IF (tx - last >= manual_timeout) AND NOT NO_AUTO_AUTO THEN
				_STATUS := 130;
			END_IF;

	132:	(* manual operation up *)
			QU := TRUE;
			QD := FALSE;
			PO := POS; AO := ANG;
			last := tx;
			IF NOT s1d.LONG THEN _STATUS := 131; dir := NOT dir; END_IF;

	133:	(* manual operation down *)
			QU := FALSE;
			QD := TRUE;
			PO := POS; AO := ANG;
			last := tx;
			IF NOT s2d.LONG THEN	_STATUS := 131; dir := NOT dir; END_IF;

	134:	(* manual operation single click up *)
			QU := TRUE;
			QD := FALSE;
			PO := POS; AO := ANG;
			IF tx - last >= max_runtime THEN _STATUS := 131; END_IF;

	135:	(* manual operation single click dn *)
			QU := FALSE;
			QD := TRUE;
			PO := POS; AO := ANG;
			IF tx - last >= max_runtime THEN _STATUS := 131;	END_IF;

	136:	(* forced input in = true *)
			QU := TRUE;
			QD := TRUE;
			PO := PI; AO := AI;
			IF tx-last >= max_runtime THEN _STATUS := 130; END_IF;

	137:	(* double click1 position *)
			QU := TRUE;
			QD := TRUE;
			PO := DBL_POS1;
			AO := DBL_ANG1;
			IF tx - last >= max_runtime THEN _STATUS := 131; END_IF;

	138:	(* double click2 position *)
			QU := TRUE;
			QD := TRUE;
			PO := DBL_POS2;
			AO := DBL_ANG2;
			IF tx - last >= max_runtime THEN _STATUS := 131; END_IF;

	   139:   (* manual operation standby *)
	         QU := FALSE;
	         QD := FALSE;
	         PO := POS;
	         AO := ANG;

END_CASE;

STATUS := _STATUS;

(* revision history
hm	29. sep 2007	rev 1.0
	original release

hm	6. oct 2007		rev 1.1
	renamed ps and as to po and ao

hm	30. dec 2007	rev 1.2
	added click_timeout variable and function

hm	16. jul. 2008	rev 1.3
	rewirtten code to allow for more functionality
	added single click mode with single_switch.
	added Debounce for inputs S1 and S2
	added double_click functionality

hm	26. sep. 2008	rev 1.4
	corrected an error while POS and ANG was transferred to outputs PO and AO during automatic modes

hm	22. jan 2009	rev 1.5
	added pulse mode for double click outputs
	added automatic mode for IN

hm	27. jul 2009	rev 1.6
	changed status 0 to 130

HF	12. nov. 2009	rev 1.7
	added state 139
	set defaults for QU, QD, PO

*)

END_FUNCTION_BLOCK

// Common/Function Blocks/DivideByN
FUNCTION_BLOCK DivideByN
VAR_INPUT
	in:BOOL;
	n:UINT;
END_VAR
VAR_OUTPUT
	out: BOOL;

END_VAR
VAR
	act:UINT;
	trigger:R_TRIG;
END_VAR

trigger(CLK:= in);
out:=FALSE;
IF NOT trigger.Q THEN RETURN; END_IF
act := act + 1;
IF act >= n THEN
	out := TRUE;
	act := 0;
END_IF

END_FUNCTION_BLOCK

// Common/Functions/AnyToUnion
FUNCTION AnyToUnion : ALL_TYPES_UNION
VAR_INPUT
	ptr:POINTER TO BYTE;
	TypeOfValue:IBaseLibrary.TypeClass;
END_VAR
VAR
END_VAR

CASE TypeOfValue OF
	IBaseLibrary.TypeClass.TYPE_SINT:
		AnyToUnion.SINT_T := TO_SINT(ptr^);
	IBaseLibrary.TypeClass.TYPE_USINT:
		AnyToUnion.USINT_T := TO_USINT(ptr^);
	IBaseLibrary.TypeClass.TYPE_INT:
		AnyToUnion.INT_T := TO_INT(ptr^);
	IBaseLibrary.TypeClass.TYPE_UINT:
		AnyToUnion.UINT_T := TO_UINT(ptr^);
	IBaseLibrary.TypeClass.TYPE_DINT:
		AnyToUnion.DINT_T := TO_DINT(ptr^);
	IBaseLibrary.TypeClass.TYPE_UDINT:
		AnyToUnion.UDINT_T := TO_UDINT(ptr^);
	IBaseLibrary.TypeClass.TYPE_LINT:
		AnyToUnion.LINT_T := TO_LINT(ptr^);
	IBaseLibrary.TypeClass.TYPE_ULINT:
		AnyToUnion.ULINT_T := TO_ULINT(ptr^);
	IBaseLibrary.TypeClass.TYPE_REAL:
		AnyToUnion.REAL_T := TO_REAL(ptr^);
	IBaseLibrary.TypeClass.TYPE_LREAL:
		AnyToUnion.LREAL_T := TO_LREAL(ptr^);
	IBaseLibrary.TypeClass.TYPE_BYTE:
		AnyToUnion.BYTE_T := TO_BYTE(ptr^);
	IBaseLibrary.TypeClass.TYPE_WORD:
		AnyToUnion.WORD_T := TO_WORD(ptr^);
	IBaseLibrary.TypeClass.TYPE_DWORD:
		AnyToUnion.DWORD_T := TO_DWORD(ptr^);
	IBaseLibrary.TypeClass.TYPE_LWORD:
		AnyToUnion.LWORD_T := TO_LWORD(ptr^);
	IBaseLibrary.TypeClass.TYPE_DATEANDTIME:
		AnyToUnion.DT_T := TO_DT(ptr^);
	IBaseLibrary.TypeClass.TYPE_TIME:
		AnyToUnion.TIME_T := TO_TIME(ptr^);
	IBaseLibrary.TypeClass.TYPE_LTIME:
		AnyToUnion.LTIME_T := TO_LTIME(ptr^);
	IBaseLibrary.TypeClass.TYPE_TIMEOFDAY:
		AnyToUnion.TOD_T := TO_TOD(ptr^);
	IBaseLibrary.TypeClass.TYPE_BOOL:
		AnyToUnion.BOOL_T := TO_BOOL(ptr^);
	IBaseLibrary.TypeClass.TYPE_DATE:
		AnyToUnion.DATE_T := TO_DATE(ptr^);
	
END_CASE

END_FUNCTION

// Common/Functions/unionToAny
FUNCTION unionToAny : BOOL
VAR_INPUT
	Value:ALL_TYPES_UNION;
	_to:POINTER TO BYTE;
	TypeOfValue:IBaseLibrary.TypeClass;
END_VAR
VAR
	Target:ALL_TYPES_UNION_POINTER;
END_VAR

Target.POINTER_TO_BYTE_T := _to;

CASE TypeOfValue OF
	IBaseLibrary.TypeClass.TYPE_SINT:
		Target.POINTER_TO_SINT_T^ := Value.SINT_T;
	IBaseLibrary.TypeClass.TYPE_USINT:
		Target.POINTER_TO_USINT_T^ := Value.USINT_T;		
	IBaseLibrary.TypeClass.TYPE_INT:
		Target.POINTER_TO_INT_T^ := Value.INT_T;
	IBaseLibrary.TypeClass.TYPE_UINT:
		Target.POINTER_TO_UINT_T^ := Value.UINT_T;
	IBaseLibrary.TypeClass.TYPE_DINT:
		Target.POINTER_TO_DINT_T^ := Value.DINT_T;
	IBaseLibrary.TypeClass.TYPE_UDINT:
		Target.POINTER_TO_UDINT_T^ := Value.UDINT_T;
	IBaseLibrary.TypeClass.TYPE_LINT:
		AtomicWriteLInt(pDest:= Target.POINTER_TO_LINT_T, liValue:= Value.LINT_T);
	IBaseLibrary.TypeClass.TYPE_ULINT:
		AtomicWriteULInt(pDest:= Target.POINTER_TO_ULINT_T, uliValue:= Value.ULINT_T);
	IBaseLibrary.TypeClass.TYPE_REAL:
		Target.POINTER_TO_REAL_T^ := Value.REAL_T;
	IBaseLibrary.TypeClass.TYPE_LREAL:
		AtomicWriteLReal(pDest:= Target.POINTER_TO_LREAL_T, lrValue:= Value.LREAL_T);
	IBaseLibrary.TypeClass.TYPE_BYTE:
		Target.POINTER_TO_BYTE_T^ := Value.BYTE_T;
	IBaseLibrary.TypeClass.TYPE_WORD:
		Target.POINTER_TO_WORD_T^ := Value.WORD_T;
	IBaseLibrary.TypeClass.TYPE_DWORD:
		Target.POINTER_TO_DWORD_T^ := Value.DWORD_T;
	IBaseLibrary.TypeClass.TYPE_LWORD:
		AtomicWriteLWord(pDest:= Target.POINTER_TO_LWORD_T, lwValue:= Value.LWORD_T);
	IBaseLibrary.TypeClass.TYPE_DATEANDTIME:
		Target.POINTER_TO_DT_T^ := Value.DT_T;
	IBaseLibrary.TypeClass.TYPE_TIME:
		Target.POINTER_TO_TIME_T^ := Value.TIME_T;
	IBaseLibrary.TypeClass.TYPE_LTIME:
		AtomicWriteLTime(pDest:= Target.POINTER_TO_LTIME_T, ltValue:= Value.LTIME_T);
	IBaseLibrary.TypeClass.TYPE_TIMEOFDAY:
		Target.POINTER_TO_TOD_T^ := Value.TOD_T;
	IBaseLibrary.TypeClass.TYPE_BOOL:
		Target.POINTER_TO_BOOL_T^ := Value.BOOL_T;
	IBaseLibrary.TypeClass.TYPE_DATE:
		Target.POINTER_TO_DATE_T^ := Value.DATE_T;
	//IBaseLibrary.TypeClass.TYPE_STRING:
		//Target.POINTER_TO_STRING_T^ := str^;
END_CASE

END_FUNCTION

// Common/Functions/checkJSON
FUNCTION checkJSON : bool
VAR_INPUT
	in:POINTER TO STRING(255);
END_VAR
VAR
	ptByte:POINTER TO BYTE;
	countOpen:UINT;
	countClose:UINT;
	textByteOpen:BYTE;
	textByteClose:BYTE;
	i:UINT;
END_VAR

i := 0;
ptByte := in;
textByteOpen := GetChar('{');
textByteClose := GetChar('}');
WHILE ptByte[i] <> 0 DO
	IF 	ptByte[i] = textByteOpen THEN countOpen := countOpen + 1;END_IF
	IF 	ptByte[i] = textByteClose THEN countClose := countClose + 1;END_IF
	i := i + 1;
END_WHILE
IF countClose <> countOpen THEN
	IF countClose > countOpen THEN
		ptByte[i - 1] := 0;
	END_IF
END_IF

END_FUNCTION
